// TIA Portal V16 export
// export: Created 2024-12-03T15:41:42.1095033Z, ExportSetting WithDefaults, DisplayName Totally Integrated Automation Portal, DisplayVersion V16 Update 6, DisplayName TIA Portal Version Control Interface, DisplayVersion V16 Update 2, DisplayName TIA Portal Openness, DisplayVersion V16 Update 6, DisplayName TIA Portal Teamcenter Gateway, DisplayVersion V16, DisplayName SINAMICS Startdrive Advanced, DisplayVersion V16 Update 5, DisplayName SINAMICS Startdrive G130, G150, S120, S150, SINAMICS MV, S210, DisplayVersion V16 Update 5, DisplayName SINAMICS Startdrive G110M, G120, G120C, G120D, G120P, G115D, DisplayVersion V16 Update 5, DisplayName STEP 7 Professional, DisplayVersion V16 Update 6, DisplayName STEP 7 Safety, DisplayVersion V16, DisplayName WinCC Advanced / Unified PC, DisplayVersion V16 Update 6
FUNCTION_BLOCK "TU_Servo_Controller_FB"   // FB85, SCL
{ S7_Optimized_Access := 'TRUE' }
VERSION : 0.1
// stored: AutoNumber true, IsIECCheckEnabled false, IsRetainMemResEnabled false, MemoryReserve 100, SetENOAutomatically false, UDAEnableTagReadback false
   VAR_INPUT
      I_DbName : String := '"Motors_Conveylinx_DB".';
      I_MotorData : "CLXAiPLC_IN_UDT";   // The 64 byte input word of the IO module
      I_ControlLeftMotorConveyLInx : Bool;   // 1 = control left motor both motos can be controlled with one module
      I_ControlRightMotorConveyLinx : Bool;   // 1 = control right motor both motors can be controlled with one fb
      I_UpFb : "SmartBooldt";   // Object is up feedback
      I_DownFb : "SmartBooldt";   // Object is down feedback
      I_TimeUp : Time := t#5s;   // time to go up
      I_TimeDown : Time := t#5s;   // time to go down
      I_Direction : Bool;   // Direction of the motor
   END_VAR
   VAR_IN_OUT
      IO_MotorStatus : "EasySystems_LineairMotor_ConveyLinx_FullPLC_Single";
      IO_MotorOutput : "CLXAiPLC_OUT_UDT";   // All the motor commands
   END_VAR
   VAR
      Sensor_UP : "SmartBool";
      Sensor_Down : "SmartBool";
      Homed { S7_SetPoint := 'True'} : "SmartBool";
      StepNumber { S7_SetPoint := 'True'} : DInt;
      PrevCmd : Real;
      S_NotConnected { S7_SetPoint := 'True'} : TON_TIME;
      S_NotUp { S7_SetPoint := 'True'} : TON_TIME;
      S_NotDown { S7_SetPoint := 'True'} : TON_TIME;
      S_srUp { S7_SetPoint := 'True'} : "SR";
      S_srDown { S7_SetPoint := 'True'} : "SR";
      CycleRun { S7_SetPoint := 'True'} : "CycleRun";
      Step_10_FindHomingPoint { S7_SetPoint := 'True'} : "StepperController";
      Step_15_ResetPulseCount { S7_SetPoint := 'True'} : "StepperController";
      Step_20_CountPulses { S7_SetPoint := 'True'} : "StepperController";
      Step_30_ResetPulseCount { S7_SetPoint := 'True'} : "StepperController";
      Step_40_RunCorrection { S7_SetPoint := 'True'} : "StepperController";
      Step_50_ResetPulseCount { S7_SetPoint := 'True'} : "StepperController";
   END_VAR
   VAR DB_SPECIFIC
      AlarmInfo { S7_SetPoint := 'True'} : "AlarmInfo_UDT";
   END_VAR
   VAR
      Overheat { S7_SetPoint := 'True'} : Program_Alarm;
      ShortCircuit { S7_SetPoint := 'True'} : Program_Alarm;
      MDRNotConnected { S7_SetPoint := 'True'} : Program_Alarm;
      Overload { S7_SetPoint := 'True'} : Program_Alarm;
      Stalled { S7_SetPoint := 'True'} : Program_Alarm;
      MDRBadHall { S7_SetPoint := 'True'} : Program_Alarm;
      OverVoltage { S7_SetPoint := 'True'} : Program_Alarm;
      LowVoltage { S7_SetPoint := 'True'} : Program_Alarm;
      NotConnected { S7_SetPoint := 'True'} : Program_Alarm;
      ConnectionNotOK { S7_SetPoint := 'True'} : Program_Alarm;
      AnyErrorActive { S7_SetPoint := 'True'} : Program_Alarm;
      JamError { S7_SetPoint := 'True'} : Program_Alarm;
      SensorLowGain { S7_SetPoint := 'True'} : Program_Alarm;
      NotUp { S7_SetPoint := 'True'} : Program_Alarm;
      NotDown { S7_SetPoint := 'True'} : Program_Alarm;
      HomingTimedOut { S7_SetPoint := 'True'} : Program_Alarm;
   END_VAR
   VAR_TEMP
      T_RunAuto : Bool;
      T_RunManual : Bool;
      T_RunInit : Bool;
      T_Setpoint : Real;
      T_AppState : "ApplicationState_UDT";
      T_ZoneInfo : "ZoneInfo";
   END_VAR
   VAR CONSTANT
      StepTimedOutHoming : DInt := 900;
   END_VAR
BEGIN
   #T_ZoneInfo := "ApplicationState_DB".ZoneNames[#IO_MotorStatus.Zone];
   #T_AppState := "ApplicationState_DB".Appstate[#T_ZoneInfo.AppStateIndex];
   #CycleRun(I_End:=15);

   REGION SENSOR INTERFACING

       #Sensor_UP(I_Sensor := #I_UpFb.State);
       #Sensor_Down(I_Sensor := #I_DownFb.State);


   END_REGION

   REGION Commands

       REGION LEFT CONTROL COMMANDS RESET
           IF #I_ControlLeftMotorConveyLInx THEN
               #IO_MotorOutput.LeftMDRControl.MDR_Direction := 0;
               #IO_MotorOutput.LeftMDRControl.Run_MDR := 0;
               #IO_MotorOutput.LeftMDRSpeed := 0;
               #IO_MotorOutput.ServoControlCommandLeft.ResetPulseCount := 0;
               #IO_MotorOutput.ServoControlCommandLeft.RunToSetpoint := 0;
               #IO_MotorOutput.LeftMDRAccel := #IO_MotorStatus.Cmd.Accel;
               #IO_MotorOutput.LeftMDRDeccel := #IO_MotorStatus.Cmd.Deaccel;
               #IO_MotorOutput.LeftMDRBrakeMode := #IO_MotorStatus.Cmd.BrakeMode;
           END_IF;
       END_REGION

       REGION RIGHT CONTROL COMMANDS RESET
           IF #I_ControlRightMotorConveyLinx THEN
               #IO_MotorOutput.RightMDRControl.MDR_Direction := 0;
               #IO_MotorOutput.RightMDRControl.Run_MDR := 0;
               #IO_MotorOutput.RightMDRSpeed := 0;
               #IO_MotorOutput.ServoControlCommandRight.ResetPulseCount := 0;
               #IO_MotorOutput.ServoControlCommandRight.RunToSetpoint := 0;
               #IO_MotorOutput.RightMDRAccel := #IO_MotorStatus.Cmd.Accel;
               #IO_MotorOutput.RightMDRDeccel := #IO_MotorStatus.Cmd.Deaccel;
               #IO_MotorOutput.RightMDRBrakeMode := #IO_MotorStatus.Cmd.BrakeMode;
           END_IF;
       END_REGION

       REGION INIT COMMANS
           #T_RunInit := 0;
       END_REGION

       REGION HOME SEQUENCE

           REGION START HOMING

               IF NOT #T_AppState.States.AutoModeActivated.State
                   AND NOT #T_AppState.States.ManualModeActivated.State THEN
                   #StepNumber := 0;
               END_IF;

               IF #T_AppState.States.AutoModeActivated.State
                   OR #T_AppState.States.ManualModeActivated.State THEN
                   IF #IO_MotorStatus.Cmd.InitPosition OR #StepNumber = 0 THEN
                       #IO_MotorStatus.Cmd.UpAuto := 0;
                       #IO_MotorStatus.Cmd.DownAuto := 0;
                       #IO_MotorStatus.Cmd.DownManual := 0;
                       #IO_MotorStatus.Cmd.UpManual := 0;
                       #StepNumber := 10;
                   END_IF;
               END_IF;

           END_REGION

           REGION STEP 10 START HOMING

               #Step_10_FindHomingPoint(I_StepNumber := 10,
                                        I_NextStepNumber := 15,
                                        I_TimeOutStepNumber := #StepTimedOutHoming,
                                        I_Condition := #Sensor_Down.O_data.LE,
                                        I_ConditionTIme := T#0ms,
                                        I_TimeOutTime := T#30s,
                                        I_PauseTimeOut := NOT #IO_MotorStatus.Status.Running,
                                        IO_StepNumber := #StepNumber);

           END_REGION

           REGION STEP 15 RESET PULSE COUNT

               #Step_15_ResetPulseCount(I_StepNumber := 15,
                                        I_NextStepNumber := 20,
                                        I_TimeOutStepNumber := #StepTimedOutHoming,
                                        I_Condition := #IO_MotorStatus.Status.ServoStatus.ResetPulseCount_Echo,
                                        I_TimeOutTime := T#5s,
                                        IO_StepNumber := #StepNumber);

           END_REGION

           REGION STEP 20 COUNT PULSES

               #Step_20_CountPulses(I_StepNumber := 20,
                                    I_NextStepNumber := 30,
                                    I_TimeOutStepNumber := #StepTimedOutHoming,
                                    I_Condition := #Sensor_Down.O_data.LE,
                                    I_ConditionTIme := t#0ms,
                                    I_TimeOutTime := T#30s,
                                    IO_StepNumber := #StepNumber);

               IF #Step_20_CountPulses.O_ConditionTrans THEN
                   #IO_MotorStatus.Settings.UpPosition := INT_TO_REAL(#IO_MotorStatus.Status.Position / 2);
               END_IF;

           END_REGION

           REGION STEP 30 RESET PULSE COUNT AFTER SECOND TWIST
               #Step_30_ResetPulseCount(I_StepNumber := 30,
                                        I_NextStepNumber := 40,
                                        I_TimeOutStepNumber := #StepTimedOutHoming,
                                        I_Condition := #IO_MotorStatus.Status.ServoStatus.ResetPulseCount_Echo,
                                        I_ConditionTIme := t#0ms,
                                        I_TimeOutTime := T#30s,
                                        IO_StepNumber := #StepNumber);

           END_REGION

           REGION STEP 40 RUN WITH CORRECTION FACTOR
               #Step_40_RunCorrection(I_StepNumber := 40,
                                      I_NextStepNumber := 50,
                                      I_TimeOutStepNumber := #StepTimedOutHoming,
                                      I_Condition := #IO_MotorStatus.Status.ServoStatus.LastServoCommandExecuted,
                                      I_ConditionTIme := t#0ms,
                                      I_TimeOutTime := T#30s,
                                      IO_StepNumber := #StepNumber);
           END_REGION

           REGION STEP 50 RESET PULSES
               #Step_50_ResetPulseCount(I_StepNumber := 50,
                                        I_NextStepNumber := 60,
                                        I_TimeOutStepNumber := #StepTimedOutHoming,
                                        I_Condition := #IO_MotorStatus.Status.ServoStatus.ResetPulseCount_Echo,
                                        I_ConditionTIme := t#0ms,
                                        I_TimeOutTime := T#30s,
                                        IO_StepNumber := #StepNumber);
           END_REGION

       END_REGION

       REGION AUTO-Manual MODE COMMANDS
           IF #T_AppState.States.AutoModeActivated.State OR #T_AppState.States.ManualModeActivated.State THEN

               REGION TWIST POSITOIN COMMANDS

                   #T_Setpoint := #PrevCmd;
                   IF #T_AppState.States.AutoModeActivated.State THEN

                       IF #IO_MotorStatus.Cmd.DownAuto THEN
                           #T_Setpoint := 0.0;
                           #IO_MotorStatus.Cmd.UpAuto := 0;
                       END_IF;

                       IF #IO_MotorStatus.Cmd.UpAuto THEN
                           #T_Setpoint := #IO_MotorStatus.Settings.UpPosition;
                           #IO_MotorStatus.Cmd.DownAuto := 0;
                       END_IF;
                   ELSE
                       #IO_MotorStatus.Cmd.UpAuto := 0;
                       #IO_MotorStatus.Cmd.DownAuto := 0;
                   END_IF;

                   IF #T_AppState.States.ManualModeActivated.State THEN

                       IF #IO_MotorStatus.Cmd.DownManual THEN
                           #T_Setpoint := 0.0;
                           #IO_MotorStatus.Cmd.UpManual := 0;
                       END_IF;

                       IF #IO_MotorStatus.Cmd.UpManual THEN
                           #T_Setpoint := #IO_MotorStatus.Settings.UpPosition;
                           #IO_MotorStatus.Cmd.DownManual := 0;
                       END_IF;
                   ELSE
                       #IO_MotorStatus.Cmd.UpManual := 0;
                       #IO_MotorStatus.Cmd.DownManual := 0;
                   END_IF;

                   IF #IO_MotorStatus.Status.Homed_Intialized THEN
                       IF NOT "CheckInRange"(I_in := #IO_MotorStatus.Status.Position, I_ReferenceValue := #T_Setpoint, I_Offset := 3) THEN
                           #IO_MotorStatus.Cmd.ServoRunToSetpoint := true;
                           #IO_MotorStatus.Cmd.ServoControlDistance := #T_Setpoint;
                       ELSE
                           #IO_MotorStatus.Cmd.ServoRunToSetpoint := FALSE;
                       END_IF;

                       IF #PrevCmd <> #T_Setpoint THEN
                           #IO_MotorStatus.Cmd.ServoRunToSetpoint := false;
                           #PrevCmd := #T_Setpoint;
                       END_IF;

                   END_IF;

               END_REGION

           END_IF;

           REGION INIT COMMANDS
               IF NOT #IO_MotorStatus.Status.Homed_Intialized THEN
                   #T_RunInit := #StepNumber = 10 OR #StepNumber = 20;
                   #IO_MotorStatus.Cmd.ServoResetPulseCount := #StepNumber = 15 OR #StepNumber = 30 OR #StepNumber = 50;
                   #IO_MotorStatus.Cmd.ServoRunToSetpoint := FALSE;
                   IF #StepNumber = 40 THEN
                       #IO_MotorStatus.Cmd.ServoRunToSetpoint := true;
                       #IO_MotorStatus.Cmd.ServoControlDistance := REAL_TO_INT(#IO_MotorStatus.Settings.PositionOffset);
                   END_IF;


                       #IO_MotorStatus.Cmd.UpAuto := 0;
                       #IO_MotorStatus.Cmd.DownAuto := 0;
                       #IO_MotorStatus.Cmd.UpManual := 0;
                       #IO_MotorStatus.Cmd.DownManual := 0;
                   END_IF;

               END_REGION

       END_REGION

       REGION INTERLOCK COMMANDS
           IF #IO_MotorStatus.Alarms.Status > 0 OR #IO_MotorStatus.Alarms.MdrAlarms.Status_1 > 0 OR #IO_MotorStatus.Status.Interlocked THEN
               #T_RunInit := 0;
               #T_Setpoint := 0;
               #IO_MotorStatus.Status.ManualCommandsDisabled := 1;
               #IO_MotorStatus.Cmd.ServoRunToSetpoint := FALSE;
           END_IF;
       END_REGION

       REGION TRANSFER LEFT COMMANDS

           IF #I_ControlLeftMotorConveyLInx THEN

               REGION DEFAULT COMMANDS
                   #IO_MotorOutput.LeftMDRControl.MDR_Direction := FALSE;
                   #IO_MotorOutput.LeftMDRAccel := #IO_MotorStatus.Cmd.Accel;

                   IF #IO_MotorStatus.Status.Homed_Intialized THEN
                       #IO_MotorOutput.LeftMDRDeccel := #IO_MotorStatus.Cmd.Deaccel;
                   ELSE
                       #IO_MotorOutput.LeftMDRDeccel := 1;
                   END_IF;

                   #IO_MotorOutput.LeftMDRBrakeMode := #IO_MotorStatus.Cmd.BrakeMode;
               END_REGION

               REGION SPEED CONTROLLER
                   IF NOT #IO_MotorStatus.Status.Homed_Intialized THEN
                       #IO_MotorOutput.LeftMDRSpeed := #IO_MotorStatus.Cmd.SpeedInit;
                   ELSE
                       #IO_MotorOutput.LeftMDRSpeed := #IO_MotorStatus.Cmd.SpeedAuto;
                   END_IF;
               END_REGION

               REGION AUTO-MANUAL MODE
                   IF #T_AppState.States.AutoModeActivated.State OR #T_AppState.States.ManualModeActivated.State THEN
                       #IO_MotorOutput.LeftMDRControl.Run_MDR := #T_RunInit;
                       #IO_MotorOutput.ServoControlCommandLeft.ResetPulseCount := #IO_MotorStatus.Cmd.ServoResetPulseCount;
                       #IO_MotorOutput.ServoControlCommandLeft.RunToSetpoint := #IO_MotorStatus.Cmd.ServoRunToSetpoint;
                       #IO_MotorOutput.ServoControlDistanceLeft := #IO_MotorStatus.Cmd.ServoControlDistance;
                   END_IF;
               END_REGION

           END_IF;

       END_REGION

       REGION TRANSFER RIGHT COMMANDS
           IF #I_ControlRightMotorConveyLinx THEN

               REGION DEFAULT COMMANDS
                   #IO_MotorOutput.RightMDRControl.MDR_Direction := FALSE;
                   #IO_MotorOutput.RightMDRAccel := #IO_MotorStatus.Cmd.Accel;

                   IF #IO_MotorStatus.Status.Homed_Intialized THEN
                       #IO_MotorOutput.RightMDRDeccel := #IO_MotorStatus.Cmd.Deaccel;
                   ELSE
                       #IO_MotorOutput.RightMDRDeccel := 1;
                   END_IF;

                   #IO_MotorOutput.RightMDRBrakeMode := #IO_MotorStatus.Cmd.BrakeMode;
               END_REGION

               REGION SPEED CONTROLLER
                   IF NOT #IO_MotorStatus.Status.Homed_Intialized THEN
                       #IO_MotorOutput.RightMDRSpeed := #IO_MotorStatus.Cmd.SpeedInit;
                   ELSE
                       #IO_MotorOutput.RightMDRSpeed := #IO_MotorStatus.Cmd.SpeedAuto;
                   END_IF;
               END_REGION

               REGION AUTO-MANUAL MODE
                   IF #T_AppState.States.AutoModeActivated.State OR #T_AppState.States.ManualModeActivated.State THEN
                       #IO_MotorOutput.RightMDRControl.Run_MDR := #T_RunInit;
                       #IO_MotorOutput.ServoControlCommandRight.ResetPulseCount := #IO_MotorStatus.Cmd.ServoResetPulseCount;
                       #IO_MotorOutput.ServoControlCommandRight.RunToSetpoint := #IO_MotorStatus.Cmd.ServoRunToSetpoint;
                       #IO_MotorOutput.ServoControlDistanceRight := #IO_MotorStatus.Cmd.ServoControlDistance;
                   END_IF;
               END_REGION

           END_IF;
       END_REGION

   END_REGION

   REGION Interlock motor

       #IO_MotorStatus.Status.Interlocked := #IO_MotorStatus.Cmd.Interlock OR NOT #T_AppState.States.EmergencyOk.State;
       #IO_MotorStatus.Status.Status.%X0 := #IO_MotorStatus.Status.Interlocked;

   END_REGION

   REGION Create status

       REGION SERVO STATUS
           #IO_MotorStatus.Status.Homed_Intialized := #StepNumber = 60;
           #Homed(I_Sensor := #IO_MotorStatus.Status.Homed_Intialized);
       END_REGION

       REGION LINEAIR POSITION STATUS

           #IO_MotorStatus.Status.PositionLineair := 0;

           //Lineair position
           IF "CheckInRange"(I_in:= #IO_MotorStatus.Status.Position,
                                      I_Offset := 10,I_ReferenceValue := #IO_MotorStatus.Settings.UpPosition)
                    AND #IO_MotorStatus.Status.Homed_Intialized
           THEN
               #IO_MotorStatus.Status.PositionLineair := 1;
           END_IF;

           IF "CheckInRange"(I_in:= #IO_MotorStatus.Status.Position,
                                 I_Offset := 10,I_ReferenceValue := 0)
               AND #IO_MotorStatus.Status.Homed_Intialized
           THEN
               #IO_MotorStatus.Status.PositionLineair := -1;
           END_IF;

       END_REGION

       REGION simulation

           IF "Simulation_DB".Simulation_On THEN
               IF #IO_MotorStatus.Cmd.UpAuto OR #IO_MotorStatus.Cmd.UpManual THEN
                   #IO_MotorStatus.Status.PositionLineair := "Up";
               END_IF;
           END_IF;

           IF "Simulation_DB".Simulation_On THEN
               IF #IO_MotorStatus.Cmd.DownAuto OR #IO_MotorStatus.Cmd.DownManual THEN
                   #IO_MotorStatus.Status.PositionLineair := "Down";
               END_IF;
           END_IF;

       END_REGION

       REGION LEFT STATUS
           IF #I_ControlLeftMotorConveyLInx THEN
               #IO_MotorStatus.Status.ActualSpeed := #I_MotorData.LeftMDRRealSpeed;
               #IO_MotorStatus.Status.Current := #I_MotorData.LeftCurrent;
               #IO_MotorStatus.Status.Frequency := #I_MotorData.LeftFreq;
               #IO_MotorStatus.Status.ManualModeActive := #IO_MotorStatus.Cmd.UpManual OR #IO_MotorStatus.Cmd.DownManual;
               #IO_MotorStatus.Status.Position := #I_MotorData.DistanceLeft;
               #IO_MotorStatus.Status.Running := #I_MotorData.LeftMDRRealSpeed > 0 AND #IO_MotorOutput.LeftMDRControl.Run_MDR;
               #IO_MotorStatus.Status.ServoStatus.LastServoCommandExecuted := #I_MotorData.ServoStatusLeft.LastServoCommandExecuted;
               #IO_MotorStatus.Status.ServoStatus.ResetPulseCount_Echo := #I_MotorData.ServoStatusLeft.ResetPulseCount_Echo;
               #IO_MotorStatus.Status.ServoStatus.RunCommand_Echo := #I_MotorData.ServoStatusLeft.RunCommand_Echo;
               #IO_MotorStatus.Status.TemperatureModule := #I_MotorData.ModuleTemp;
               #IO_MotorStatus.Status.TeperatureMDR := #I_MotorData.LeftCalcTemp;
           END_IF;
       END_REGION

       REGION RIGHT STATUS
           IF #I_ControlRightMotorConveyLinx THEN
               #IO_MotorStatus.Status.ActualSpeed := #I_MotorData.RightMDRRealSpeed;
               #IO_MotorStatus.Status.Current := #I_MotorData.RightCurrent;
               #IO_MotorStatus.Status.Frequency := #I_MotorData.RightFreq;
               #IO_MotorStatus.Status.ManualModeActive := #IO_MotorStatus.Cmd.UpManual OR #IO_MotorStatus.Cmd.DownManual;
               #IO_MotorStatus.Status.Position := #I_MotorData.DistanceRight;
               #IO_MotorStatus.Status.Running := #I_MotorData.RightMDRRealSpeed > 0 AND #IO_MotorOutput.RightMDRControl.Run_MDR;
               #IO_MotorStatus.Status.ServoStatus.LastServoCommandExecuted := #I_MotorData.ServoStatusRight.LastServoCommandExecuted;
               #IO_MotorStatus.Status.ServoStatus.ResetPulseCount_Echo := #I_MotorData.ServoStatusRight.ResetPulseCount_Echo;
               #IO_MotorStatus.Status.ServoStatus.RunCommand_Echo := #I_MotorData.ServoStatusRight.RunCommand_Echo;
               #IO_MotorStatus.Status.TemperatureModule := #I_MotorData.ModuleTemp;
               #IO_MotorStatus.Status.TeperatureMDR := #I_MotorData.RightCalcTemp;
           END_IF;
       END_REGION

       REGION Min max voltage

           #IO_MotorStatus.Status.Voltage := #I_MotorData.Voltage;
           IF #I_MotorData.Voltage < #IO_MotorStatus.Status.MinVoltage THEN
               #IO_MotorStatus.Status.MinVoltage := #I_MotorData.Voltage;
           END_IF;

           IF #I_MotorData.Voltage > #IO_MotorStatus.Status.MaxVoltage THEN
               #IO_MotorStatus.Status.MaxVoltage := #I_MotorData.Voltage;
           END_IF;

       END_REGION

       #IO_MotorStatus.Status.ManualModeActive := #T_AppState.States.ManualModeActivated.State;
       #IO_MotorStatus.Status.Status.%X1 := #IO_MotorStatus.Status.Running;
       #IO_MotorStatus.Status.Status.%X2 := #IO_MotorStatus.Status.ManualModeActive;

   END_REGION

   REGION Check alarm active

       IF #I_ControlLeftMotorConveyLInx THEN

           IF #I_MotorData.LeftMDRDiagnostic.LowVoltage THEN
               #IO_MotorStatus.Alarms.MdrAlarms.LowVoltage.Active := True;
           END_IF;

           IF #I_MotorData.LeftMDRDiagnostic.MDRBadHall THEN
               #IO_MotorStatus.Alarms.MdrAlarms.MDRBadHall.Active := True;
           END_IF;

           IF #I_MotorData.LeftMDRDiagnostic.MDRNotConnected THEN
               #IO_MotorStatus.Alarms.MdrAlarms.MDRNotConnected.Active := True;
           END_IF;

           IF #I_MotorData.LeftMDRDiagnostic.Overheat THEN
               #IO_MotorStatus.Alarms.MdrAlarms.Overheat.Active := True;
           END_IF;

           IF #I_MotorData.LeftMDRDiagnostic.Overload THEN
               #IO_MotorStatus.Alarms.MdrAlarms.Overload.Active := True;
           END_IF;

           IF #I_MotorData.LeftMDRDiagnostic.OverVoltage THEN
               #IO_MotorStatus.Alarms.MdrAlarms.OverVoltage.Active := True;
           END_IF;

           IF #I_MotorData.LeftMDRDiagnostic.ShortCircuit THEN
               #IO_MotorStatus.Alarms.MdrAlarms.ShortCircuit.Active := True;
           END_IF;

           IF #I_MotorData.LeftMDRDiagnostic.Stalled THEN
               #IO_MotorStatus.Alarms.MdrAlarms.Stalled.Active := True;
           END_IF;

       END_IF;

       IF #I_ControlRightMotorConveyLinx THEN

           IF #I_MotorData.RightMDRDiagnostic.LowVoltage THEN
               #IO_MotorStatus.Alarms.MdrAlarms.LowVoltage.Active := True;
           END_IF;

           IF #I_MotorData.RightMDRDiagnostic.MDRBadHall THEN
               #IO_MotorStatus.Alarms.MdrAlarms.MDRBadHall.Active := True;
           END_IF;

           IF #I_MotorData.RightMDRDiagnostic.MDRNotConnected THEN
               #IO_MotorStatus.Alarms.MdrAlarms.MDRNotConnected.Active := True;
           END_IF;

           IF #I_MotorData.RightMDRDiagnostic.Overheat THEN
               #IO_MotorStatus.Alarms.MdrAlarms.Overheat.Active := True;
           END_IF;

           IF #I_MotorData.RightMDRDiagnostic.Overload THEN
               #IO_MotorStatus.Alarms.MdrAlarms.Overload.Active := True;
           END_IF;

           IF #I_MotorData.RightMDRDiagnostic.OverVoltage THEN
               #IO_MotorStatus.Alarms.MdrAlarms.OverVoltage.Active := True;
           END_IF;

           IF #I_MotorData.RightMDRDiagnostic.ShortCircuit THEN
               #IO_MotorStatus.Alarms.MdrAlarms.ShortCircuit.Active := True;
           END_IF;

           IF #I_MotorData.RightMDRDiagnostic.Stalled THEN
               #IO_MotorStatus.Alarms.MdrAlarms.Stalled.Active := True;
           END_IF;

       END_IF;

       #IO_MotorStatus.Heartbeat := #I_MotorData.AllSensors.Heartbeat;
       #S_NotConnected(IN := NOT #IO_MotorStatus.Heartbeat,
                       PT := t#5s);

       IF #S_NotConnected.Q THEN
           #IO_MotorStatus.Alarms.MdrAlarms.NotConnected.Active := true;
       END_IF;

       //Not up
       #S_NotUp(IN := (#IO_MotorStatus.Cmd.UpAuto OR #IO_MotorStatus.Cmd.UpManual)
                AND  #IO_MotorStatus.Status.PositionLineair <> 1
                AND #IO_MotorStatus.Status.Homed_Intialized,
                PT := #I_TimeUp);

       IF #S_NotUp.Q THEN
           #IO_MotorStatus.Alarms.NotUp.Active := true;
       END_IF;

       //Not down
       #S_NotDown(IN := (#IO_MotorStatus.Cmd.DownAuto OR #IO_MotorStatus.Cmd.DownManual)
                  AND #IO_MotorStatus.Status.PositionLineair <> -1
                  AND #IO_MotorStatus.Status.Homed_Intialized,
                  PT := #I_TimeDown);

       IF #S_NotDown.Q THEN
           #IO_MotorStatus.Alarms.NotDown.Active := true;
       END_IF;

       REGION HOMING TIMED OUT
           IF #StepNumber = #StepTimedOutHoming THEN
               #IO_MotorStatus.Alarms.HomingTimedOut.Active := true;
           END_IF;
       END_REGION

       REGION PROGRAM ALARMS

           REGION alarm info
               IF "HMI_DB".ReloadSettings.signal OR NOT #AlarmInfo.init OR #AlarmInfo.info = '' OR #IO_MotorStatus.Info.Name = '' THEN
                   #IO_MotorStatus.Info.Name := "buildObjectName"(I_Symbolname := GetSymbolName(variable := #IO_MotorStatus, size:=100));
                   #AlarmInfo.info := "buildAlarmInfo"(I_ZoneIndex := #IO_MotorStatus.Zone, I_ZoneName := #T_ZoneInfo.ZoneName, I_ObjectName := #IO_MotorStatus.Info.Name);
                   #AlarmInfo.init := TRUE;
               END_IF;
           END_REGION

           REGION PROGRAM ALARMS MDR

               IF #CycleRun.O_Cycle = 1 THEN
                   #Overheat(SIG := #IO_MotorStatus.Alarms.MdrAlarms.Overheat.Active,
                             SD_1 := #T_ZoneInfo.ZoneName,
                             SD_2 := #IO_MotorStatus.Info.Name,
                             SD_3 := #AlarmInfo.info);
               END_IF;

               IF #CycleRun.O_Cycle = 2 THEN
                   #ShortCircuit(SIG := #IO_MotorStatus.Alarms.MdrAlarms.ShortCircuit.Active,
                                 SD_1 := #T_ZoneInfo.ZoneName,
                                 SD_2 := #IO_MotorStatus.Info.Name,
                                 SD_3 := #AlarmInfo.info);
               END_IF;

               IF #CycleRun.O_Cycle = 3 THEN
                   #MDRNotConnected(SIG := #IO_MotorStatus.Alarms.MdrAlarms.MDRNotConnected.Active,
                                    SD_1 := #T_ZoneInfo.ZoneName,
                                    SD_2 := #IO_MotorStatus.Info.Name,
                                    SD_3 := #AlarmInfo.info);
               END_IF;

               IF #CycleRun.O_Cycle = 4 THEN
                   #Overload(SIG := #IO_MotorStatus.Alarms.MdrAlarms.Overload.Active,
                             SD_1 := #T_ZoneInfo.ZoneName,
                             SD_2 := #IO_MotorStatus.Info.Name,
                             SD_3 := #AlarmInfo.info);
               END_IF;

               IF #CycleRun.O_Cycle = 5 THEN
                   #Stalled(SIG := #IO_MotorStatus.Alarms.MdrAlarms.Stalled.Active,
                            SD_1 := #T_ZoneInfo.ZoneName,
                            SD_2 := #IO_MotorStatus.Info.Name,
                            SD_3 := #AlarmInfo.info);
               END_IF;

               IF #CycleRun.O_Cycle = 6 THEN
                   #MDRBadHall(SIG := #IO_MotorStatus.Alarms.MdrAlarms.MDRBadHall.Active,
                               SD_1 := #T_ZoneInfo.ZoneName,
                               SD_2 := #IO_MotorStatus.Info.Name,
                               SD_3 := #AlarmInfo.info);
               END_IF;

                   IF #CycleRun.O_Cycle = 7 THEN
                       #OverVoltage(SIG := #IO_MotorStatus.Alarms.MdrAlarms.OverVoltage.Active,
                                    SD_1 := #T_ZoneInfo.ZoneName,
                                    SD_2 := #IO_MotorStatus.Info.Name,
                                    SD_3 := #AlarmInfo.info);
                   END_IF;

                   IF #CycleRun.O_Cycle = 8 THEN
                       #LowVoltage(SIG := #IO_MotorStatus.Alarms.MdrAlarms.LowVoltage.Active,
                                   SD_1 := #T_ZoneInfo.ZoneName,
                                   SD_2 := #IO_MotorStatus.Info.Name,
                                   SD_3 := #AlarmInfo.info);
                   END_IF;

                   IF #CycleRun.O_Cycle = 9 THEN
                       #NotConnected(SIG := #IO_MotorStatus.Alarms.MdrAlarms.NotConnected.Active,
                                     SD_1 := #T_ZoneInfo.ZoneName,
                                     SD_2 := #IO_MotorStatus.Info.Name,
                                     SD_3 := #AlarmInfo.info);
                   END_IF;

                   IF #CycleRun.O_Cycle = 10 THEN
                       #ConnectionNotOK(SIG := #IO_MotorStatus.Alarms.MdrAlarms.ConnectionNotOK.Active,
                                        SD_1 := #T_ZoneInfo.ZoneName,
                                        SD_2 := #IO_MotorStatus.Info.Name,
                                        SD_3 := #AlarmInfo.info);
                   END_IF;

                   IF #CycleRun.O_Cycle = 11 THEN
                       #AnyErrorActive(SIG := #IO_MotorStatus.Alarms.MdrAlarms.AnyErrorActive.Active,
                                       SD_1 := #T_ZoneInfo.ZoneName,
                                       SD_2 := #IO_MotorStatus.Info.Name,
                                       SD_3 := #AlarmInfo.info);
                   END_IF;

                   IF #CycleRun.O_Cycle = 12 THEN
                       #JamError(SIG := #IO_MotorStatus.Alarms.MdrAlarms.JamError.Active,
                                 SD_1 := #T_ZoneInfo.ZoneName,
                                 SD_2 := #IO_MotorStatus.Info.Name,
                                 SD_3 := #AlarmInfo.info);
                   END_IF;

                   IF #CycleRun.O_Cycle = 13 THEN
                       #SensorLowGain(SIG := #IO_MotorStatus.Alarms.MdrAlarms.SensorLowGain.Active,
                                      SD_1 := #T_ZoneInfo.ZoneName,
                                      SD_2 := #IO_MotorStatus.Info.Name,
                                      SD_3 := #AlarmInfo.info);
                   END_IF;

           END_REGION

           REGION PROGRAM ALARMS TRANSFER UNIT

               IF #CycleRun.O_Cycle = 14 THEN
                   #NotUp(SIG := #IO_MotorStatus.Alarms.NotUp.Active,
                          SD_1 := #T_ZoneInfo.ZoneName,
                          SD_2 := #IO_MotorStatus.Info.Name,
                          SD_3 := #AlarmInfo.info);
               END_IF;

               IF #CycleRun.O_Cycle = 15 THEN
                   #NotDown(SIG := #IO_MotorStatus.Alarms.NotDown.Active,
                            SD_1 := #T_ZoneInfo.ZoneName,
                            SD_2 := #IO_MotorStatus.Info.Name,
                            SD_3 := #AlarmInfo.info);

                   #HomingTimedOut(SIG := #IO_MotorStatus.Alarms.HomingTimedOut.Active,
                            SD_1 := #T_ZoneInfo.ZoneName,
                            SD_2 := #IO_MotorStatus.Info.Name,
                            SD_3 := #AlarmInfo.info);

               END_IF;


           END_REGION

       END_REGION

   END_REGION

   REGION Alarm status

       #IO_MotorStatus.Alarms.Status.%X0 := #IO_MotorStatus.Alarms.NotUp.Active;
       #IO_MotorStatus.Alarms.Status.%X1 := #IO_MotorStatus.Alarms.NotDown.Active;
       #IO_MotorStatus.Alarms.Status.%X2 := #IO_MotorStatus.Alarms.HomingTimedOut.Active;
       #IO_MotorStatus.Alarms.Status.%X3 := #IO_MotorStatus.Alarms.MdrAlarms.Status_1 > 0;

       REGION MDR alarms

           #IO_MotorStatus.Alarms.MdrAlarms.Status_1.%X0 := #IO_MotorStatus.Alarms.MdrAlarms.Overheat.Active;
           //#MotorStatus.Alarms.MdrAlarms.Status_1.%X1 := #MotorStatus.Alarms.MdrAlarms.Overheat.Active;
           #IO_MotorStatus.Alarms.MdrAlarms.Status_1.%X2 := #IO_MotorStatus.Alarms.MdrAlarms.ShortCircuit.Active;
           #IO_MotorStatus.Alarms.MdrAlarms.Status_1.%X3 := #IO_MotorStatus.Alarms.MdrAlarms.MDRNotConnected.Active;

           #IO_MotorStatus.Alarms.MdrAlarms.Status_1.%X4 := #IO_MotorStatus.Alarms.MdrAlarms.Overload.Active;
           #IO_MotorStatus.Alarms.MdrAlarms.Status_1.%X5 := #IO_MotorStatus.Alarms.MdrAlarms.Stalled.Active;
           #IO_MotorStatus.Alarms.MdrAlarms.Status_1.%X6 := #IO_MotorStatus.Alarms.MdrAlarms.MDRBadHall.Active;
           // #MotorStatus.Alarms.MdrAlarms.Status_1.%X7 := #MotorStatus.Alarms.MdrAlarms.Overheat.Active;

           #IO_MotorStatus.Alarms.MdrAlarms.Status_1.%X8 := #IO_MotorStatus.Alarms.MdrAlarms.OverVoltage.Active;
           #IO_MotorStatus.Alarms.MdrAlarms.Status_1.%X9 := #IO_MotorStatus.Alarms.MdrAlarms.LowVoltage.Active;
           #IO_MotorStatus.Alarms.MdrAlarms.Status_1.%X10 := #IO_MotorStatus.Alarms.MdrAlarms.NotConnected.Active;
           #IO_MotorStatus.Alarms.MdrAlarms.Status_1.%X11 := #IO_MotorStatus.Alarms.MdrAlarms.ConnectionNotOK.Active;

           #IO_MotorStatus.Alarms.MdrAlarms.Status_1.%X12 := #IO_MotorStatus.Alarms.MdrAlarms.AnyErrorActive.Active;
           #IO_MotorStatus.Alarms.MdrAlarms.Status_1.%X13 := #IO_MotorStatus.Alarms.MdrAlarms.JamError.Active;
           #IO_MotorStatus.Alarms.MdrAlarms.Status_1.%X14 := #IO_MotorStatus.Alarms.MdrAlarms.SensorLowGain.Active;
           #IO_MotorStatus.Alarms.MdrAlarms.Status_1.%X15 := #IO_MotorStatus.Alarms.MdrAlarms.Overheat.Active;

       END_REGION

       IF #IO_MotorStatus.Alarms.Status > 0 THEN
           "ApplicationState_DB".Appstate[#T_ZoneInfo.AppStateIndex].Alarms.AlarmActiveInternalPLC := TRUE;
       END_IF;

   END_REGION

   REGION Reset alarms

       IF (#IO_MotorStatus.Alarms.Status > 0 AND (#T_AppState.Hmi_Buttons.reset.state.State OR #IO_MotorStatus.Cmd.Reset))
           OR #IO_MotorStatus.Cmd.InitPosition
           OR "Simulation_DB".Simulation_On THEN

           #IO_MotorStatus.Alarms.MdrAlarms.Overheat.Active := False;
           #IO_MotorStatus.Alarms.MdrAlarms.Overheat.Active := False;
           #IO_MotorStatus.Alarms.MdrAlarms.ShortCircuit.Active := False;
           #IO_MotorStatus.Alarms.MdrAlarms.MDRNotConnected.Active := False;

           #IO_MotorStatus.Alarms.MdrAlarms.Overload.Active := False;
           #IO_MotorStatus.Alarms.MdrAlarms.Stalled.Active := False;
           #IO_MotorStatus.Alarms.MdrAlarms.MDRBadHall.Active := False;
           #IO_MotorStatus.Alarms.MdrAlarms.Overheat.Active := False;
           #IO_MotorStatus.Alarms.MdrAlarms.OverVoltage.Active := False;
           #IO_MotorStatus.Alarms.MdrAlarms.LowVoltage.Active := False;
           #IO_MotorStatus.Alarms.MdrAlarms.NotConnected.Active := False;
           #IO_MotorStatus.Alarms.MdrAlarms.ConnectionNotOK.Active := False;

           #IO_MotorStatus.Alarms.MdrAlarms.AnyErrorActive.Active := False;
           #IO_MotorStatus.Alarms.MdrAlarms.JamError.Active := False;
           #IO_MotorStatus.Alarms.MdrAlarms.SensorLowGain.Active := False;
           #IO_MotorStatus.Alarms.MdrAlarms.Overheat.Active := False;

           #IO_MotorStatus.Alarms.NotDown.Active := 0;
           #IO_MotorStatus.Alarms.NotUp.Active := 0;
           #IO_MotorStatus.Alarms.HomingTimedOut.Active := 0;
           #StepNumber := 0;

           #IO_MotorStatus.Alarms.Status := 0;
           #IO_MotorStatus.Alarms.MdrAlarms.Status_1 := 0;

       END_IF;

   END_REGION

   REGION common status
       #IO_MotorStatus.Info.CommonStatus := 0;
       IF #IO_MotorStatus.Status.Running THEN
           #IO_MotorStatus.Info.CommonStatus := 1;
       END_IF;

       IF #IO_MotorStatus.Alarms.Status > 1 THEN
           #IO_MotorStatus.Info.CommonStatus := -1;
       END_IF;
   END_REGION

   IF #IO_MotorStatus.Cmd.InitPosition THEN
       #IO_MotorStatus.Cmd.InitPosition := FALSE;
   END_IF;

   IF #IO_MotorStatus.Cmd.Reset THEN
       #IO_MotorStatus.Cmd.Reset := FALSE;
   END_IF;
END_FUNCTION_BLOCK
